Staubli VAL3: pick.pgx

program pick(num x_nX, num x_nY)
begin



  pPick.trsf.x = x_nX*100
  pPick.trsf.y = x_nY*100

  movej(appro(pPick,trApro),tGreifer, mUsedSpeed)
  movel(pPick, tGreifer, mUsedSpeed)
  close(tGreifer)
  movel(appro(pPick, trApro), tGreifer, mUsedSpeed)
  logMsg("Objekt aufgegriffen")





end
